// TIA Portal V19 export
DATA_BLOCK "PublishedDB"   // DB3
// stored: Access Published, MemoryReserve 100, Namespace Unit3
   VAR
      req : "Unit3.type_u3RequestData";
      response { S7_SetPoint := 'True'} : "Unit3.type_u3ResponsetData";
      u3ToXyz { S7_SetPoint := 'True'} : "Unit3.type_u3ToXyz";
      xyzToU3 { S7_SetPoint := 'True'} : "Unit3.type_XyzToU3";
      ngConveyorToU2Handlingxyz { S7_SetPoint := 'True'} : "LEXCHANGETRAY_typeNgConveyorEm_interface";
      ngConveyorToU1Handlingxyz { S7_SetPoint := 'True'} : "LEXCHANGETRAY_typeNgConveyorEm_interface";
   END_VAR
BEGIN
END_DATA_BLOCK
